Fanuc KAREL source: mth_pow.kl

PROGRAM mth_pow
%NOBUSYLAMP
%NOLOCKGROUP

VAR
	out_reg : INTEGER
	value : REAL
	exponent : REAL
%from tpe.klh %import get_int_arg,get_real_arg
%from registers.klh %import set_real
%from math.klh %import pow

BEGIN
	value = tpe__get_real_arg(1)
	exponent = tpe__get_real_arg(2)
	out_reg = tpe__get_int_arg(3)
	registers__set_real(out_reg, math__pow(value,exponent))
END mth_pow
